{attribute 'OPC.UA.DA.StructuredType' := '1'}
TYPE stCmd :
STRUCT
	iCmd	: INT;	(* Codice comando *)
	iPar1	: INT;	(* Parametro 1 *)
	iPar2	: INT;	(* Parametro 2 *)
END_STRUCT
END_TYPE

(* stored: Version 1.1.0.1, ProductVersion 3.1.4024.11
   DUT stCmd: Id {cf3ea72b-51fb-47db-a51b-41f1bee5ea84} *)
